FUNCTION_BLOCK FB_MUX_LINT (* See FB_MUX_ANY *)
  (* Standard: IEC 61499 *)
  (* Version 0.1, 2006-09-13, JHC, Holobloc Inc, Moved to fb.rt.select. *)
  (* Version 0.0, 2004-12-15, JHC, Rockwell Automation, Converted from SRC format. *)
  (* Compiler header: package fb.rt.select; *)
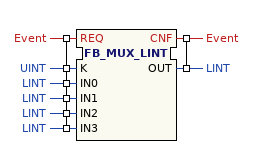
  EVENT_INPUT
    REQ WITH K, IN0, IN1, IN2, IN3;
  END_EVENT
  EVENT_OUTPUT
    CNF WITH OUT;
  END_EVENT
  VAR_INPUT
    K : UINT;
    IN0 : LINT;
    IN1 : LINT;
    IN2 : LINT;
    IN3 : LINT;
  END_VAR
  VAR_OUTPUT
    OUT : LINT;
  END_VAR
END_FUNCTION_BLOCK
